# EPICS substitutions: ADApp/Db/NDRoiStatNDims.substitutions
file "NDDims.template"
{
    pattern { DIM, MIN_PARAM,         SIZE_PARAM,        ADDR,         TIMEOUT }
            { X,   ROISTAT_DIM0_MIN,  ROISTAT_DIM0_SIZE, "\$(ADDR=0)", "\$(TIMEOUT=1)" }
            { Y,   ROISTAT_DIM1_MIN,  ROISTAT_DIM1_SIZE, "\$(ADDR=0)", "\$(TIMEOUT=1)" }
}
